(* IEC 61131-3 sources: vscode-st/examples, 13 files *)

(* ---- 02-function.st ---- *)
/* 02-function.st — FUNCTION with return type

   Demonstrates FUNCTION declaration with VAR_INPUT, local VAR, return value,
   RETURN statement (early exit), and function body with expressions. */

FUNCTION AddValues : INT
VAR_INPUT
    a : INT;
    b : INT;
END_VAR
VAR
    temp : INT;
END_VAR

// Compute sum and return
temp := a + b;

// Early RETURN guard — skips rest if condition met
IF temp > 1000 THEN
    AddValues := 0;
    RETURN;
END_IF;

AddValues := temp;

END_FUNCTION

(* ---- 03-function-block.st ---- *)
/* 03-function-block.st — FUNCTION_BLOCK

   Demonstrates FUNCTION_BLOCK with VAR_INPUT, VAR_OUTPUT, VAR,
   internal state logic, and ACTION definitions. */

FUNCTION_BLOCK CounterFB
VAR_INPUT
    enable  : BOOL;
    reset   : BOOL;
    maxVal  : INT := 100;
END_VAR
VAR_OUTPUT
    overflow : BOOL;
    current  : INT;
END_VAR
VAR
    internal : INT;
END_VAR

IF reset THEN
    internal := 0;
    current  := 0;
    overflow := FALSE;
ELSIF enable THEN
    IF internal < maxVal THEN
        internal := internal + 1;
    ELSE
        overflow := TRUE;
    END_IF;
    current := internal;
END_IF;

END_FUNCTION_BLOCK

FUNCTION_BLOCK MotorWithActions
VAR_INPUT
    startCmd : BOOL;
    stopCmd  : BOOL;
    speed    : REAL;
END_VAR
VAR_OUTPUT
    running    : BOOL;
    currentRPM : REAL;
END_VAR
VAR
    rampStep : REAL := 10.0;
END_VAR

IF startCmd THEN
    StartRamp();
ELSIF stopCmd THEN
    StopRamp();
END_IF;

ACTION StartRamp
    IF NOT running THEN
        running := TRUE;
        currentRPM := 0.0;
    END_IF;
    IF currentRPM < speed THEN
        currentRPM := currentRPM + rampStep;
    END_IF;
END_ACTION

ACTION StopRamp
    IF currentRPM > 0.0 THEN
        currentRPM := currentRPM - rampStep;
    ELSE
        running := FALSE;
        currentRPM := 0.0;
    END_IF;
END_ACTION

END_FUNCTION_BLOCK

(* ---- 04-namespace.st ---- *)
/* 04-namespace.st — NAMESPACE

   Demonstrates NAMESPACE containing multiple POU definitions.
   Namespaces group related POUs and provide name scoping. */

NAMESPACE MotorControl

    FUNCTION CalculateSpeed : REAL
    VAR_INPUT
        rpm     : INT;
        gearRatio : REAL;
    END_VAR
    VAR
        result : REAL;
    END_VAR
    result := INT_TO_REAL(rpm) * gearRatio;
    CalculateSpeed := result;
    END_FUNCTION

    PROGRAM MotorRunner
    VAR
        speed   : REAL;
        running : BOOL;
    END_VAR
    speed := CalculateSpeed(rpm := 1500, gearRatio := 3.14);
    IF running THEN
        speed := speed * 1.05;
    END_IF;
    END_PROGRAM

    FUNCTION_BLOCK PIDController
    VAR_INPUT
        setpoint : REAL;
        actual   : REAL;
        kp       : REAL := 1.0;
    END_VAR
    VAR_OUTPUT
        output : REAL;
    END_VAR
    VAR
        error : REAL;
    END_VAR
    error := setpoint - actual;
    output := kp * error;
    END_FUNCTION_BLOCK

END_NAMESPACE

(* ---- 06-class.st ---- *)
/* 06-class.st — CLASS, METHOD, PROPERTY (IEC 61131-3 OOP)

   Demonstrates CLASS declarations with access modifiers (PUBLIC, PRIVATE,
   PROTECTED, INTERNAL), ABSTRACT/FINAL/OVERRIDE method modifiers,
   PROPERTY with GET/SET, EXTENDS, and IMPLEMENTS. */

CLASS MotorBase IMPLEMENTS IMotor
    VAR
        _speed    : REAL;
        _enabled  : BOOL;
        _name     : STRING := 'MotorBase';
    END_VAR

    METHOD PUBLIC Start : BOOL
        _enabled := TRUE;
        Start := TRUE;
    END_METHOD

    METHOD PUBLIC Stop : BOOL
        _enabled := FALSE;
        _speed := 0.0;
        Stop := TRUE;
    END_METHOD

    METHOD PUBLIC SetSpeed : BOOL
    VAR_INPUT
        newSpeed : REAL;
    END_VAR
        IF _enabled THEN
            _speed := LIMIT(0.0, newSpeed, _maxSpeed);
            SetSpeed := TRUE;
        ELSE
            SetSpeed := FALSE;
        END_IF;
    END_METHOD

    METHOD PROTECTED GetMaxSpeed : REAL
        GetMaxSpeed := _maxSpeed;
    END_METHOD

END_CLASS

CLASS AdvancedMotor EXTENDS MotorBase IMPLEMENTS IAdvancedMotor
    VAR PRIVATE
        _accelRate : REAL := 5.0;
        _decelRate : REAL := 10.0;
        _targetSpeed : REAL;
    END_VAR

    VAR PUBLIC
        status : STRING := 'idle';
    END_VAR

    // Override the Start method
    METHOD PUBLIC OVERRIDE Start : BOOL
        status := 'ramping';
        Start := SUPER.Start();
    END_METHOD

    // Abstract method that must be implemented
    METHOD PUBLIC ABSTRACT Diagnose : STRING
    END_METHOD

    METHOD PUBLIC FINAL GetConfig : STRING
        GetConfig := CONCAT('Motor: ', _name);
    END_METHOD

    // Property with getter and setter
    PROPERTY PUBLIC TargetSpeed : REAL
        GET
            TargetSpeed := _targetSpeed;
        END_GET
        SET
            _targetSpeed := LIMIT(0.0, TargetSpeed, SUPER.GetMaxSpeed());
        END_SET
    END_PROPERTY

    // Read-only property (getter only)
    PROPERTY PUBLIC IsRunning : BOOL
        GET
            IsRunning := _enabled AND (_speed > 0.0);
        END_GET
    END_PROPERTY

    METHOD INTERNAL RampToTarget : BOOL
        IF _speed < _targetSpeed THEN
            _speed := _speed + _accelRate;
            IF _speed > _targetSpeed THEN
                _speed := _targetSpeed;
            END_IF;
        ELSIF _speed > _targetSpeed THEN
            _speed := _speed - _decelRate;
            IF _speed < _targetSpeed THEN
                _speed := _targetSpeed;
            END_IF;
        END_IF;
        status := CONCAT('speed: ', REAL_TO_STRING(_speed));
        RampToTarget := TRUE;
    END_METHOD

END_CLASS

(* ---- 07-interface.st ---- *)
/* 07-interface.st — INTERFACE with METHOD signatures

   Demonstrates INTERFACE declarations with METHOD signatures (no body)
   and IMPLEMENTS relationship with CLASS / FUNCTION_BLOCK. */

INTERFACE IMotor
    METHOD Start : BOOL
    END_METHOD

    METHOD Stop : BOOL
    END_METHOD

    METHOD SetSpeed : BOOL
    VAR_INPUT
        newSpeed : REAL;
    END_VAR
    END_METHOD

    METHOD GetName : STRING
    END_METHOD
END_INTERFACE

INTERFACE IAdvancedMotor EXTENDS IMotor
    METHOD Diagnose : STRING
    END_METHOD

    METHOD GetEfficiency : REAL
    VAR_INPUT
        loadPercent : INT;
    END_VAR
    END_METHOD

    METHOD EmergencyStop : BOOL
    END_METHOD
END_INTERFACE

INTERFACE ISerializable
    METHOD Serialize : STRING
    END_METHOD

    METHOD Deserialize : BOOL
    VAR_IN_OUT
        data : STRING;
    END_VAR
    END_METHOD
END_INTERFACE

// A function block implementing multiple interfaces
FUNCTION_BLOCK SmartMotor IMPLEMENTS IAdvancedMotor, ISerializable
    VAR
        _speed       : REAL;
        _enabled     : BOOL;
        _serialized  : STRING;
    END_VAR

    METHOD PUBLIC Start : BOOL
        _enabled := TRUE;
        Start := TRUE;
    END_METHOD

    METHOD PUBLIC Stop : BOOL
        _enabled := FALSE;
        _speed := 0.0;
        Stop := TRUE;
    END_METHOD

    METHOD PUBLIC SetSpeed : BOOL
    VAR_INPUT
        newSpeed : REAL;
    END_VAR
        _speed := newSpeed;
        SetSpeed := TRUE;
    END_METHOD

    METHOD PUBLIC GetName : STRING
        GetName := 'SmartMotor';
    END_METHOD

    METHOD PUBLIC Diagnose : STRING
        Diagnose := CONCAT('Speed=', REAL_TO_STRING(_speed));
    END_METHOD

    METHOD PUBLIC GetEfficiency : REAL
    VAR_INPUT
        loadPercent : INT;
    END_VAR
        GetEfficiency := 0.85;
    END_METHOD

    METHOD PUBLIC EmergencyStop : BOOL
        _enabled := FALSE;
        _speed := 0.0;
        EmergencyStop := TRUE;
    END_METHOD

    METHOD PUBLIC Serialize : STRING
        Serialize := CONCAT('SmartMotor:', REAL_TO_STRING(_speed));
    END_METHOD

    METHOD PUBLIC Deserialize : BOOL
    VAR_IN_OUT
        data : STRING;
    END_VAR
        Deserialize := TRUE;
    END_METHOD

END_FUNCTION_BLOCK

(* ---- 10-var-blocks.st ---- *)
/* 10-var-blocks.st — All VAR block variants

   Demonstrates every VAR keyword variant from the grammar: VAR, VAR_INPUT,
   VAR_OUTPUT, VAR_IN_OUT, VAR_GLOBAL with qualifiers (RETAIN, PERSISTENT,
   CONSTANT), AT addresses, comma-separated declarations, and VAR_EXTERNAL
   inside a POU. */

// Global variable block — available across the project
VAR_GLOBAL
    gSystemTick  : DINT;
    gMaxSpeed    : REAL    := 5000.0;
    gMachineName : STRING  := 'PLC001';
END_VAR

// Retained global — survives power cycle
VAR_GLOBAL RETAIN
    gRuntimeHours : DINT;
    gCycleCount   : DWORD;
END_VAR

// Persistent global — survives cold reset
VAR_GLOBAL PERSISTENT
    gSerialNumber : STRING  := 'SN-0001';
    gCalibration  : REAL    := 1.0;
END_VAR

// Constant global
VAR_GLOBAL CONSTANT
    gPI           : REAL    := 3.14159265359;
    gMaxMotors    : INT     := 8;
    gVersion      : STRING  := 'v2.0.0';
END_VAR

FUNCTION_BLOCK VarBlockDemo
    // Standard local variables
    VAR
        localCounter : INT;
        localFlag    : BOOL;
    END_VAR

    // Temporary — not retained across cycles
    VAR
        tempCalc     : REAL;
        tempString   : STRING;
    END_VAR

    // Input variables
    VAR_INPUT
        inEnable      : BOOL;
        inSpeedRef    : REAL;
    END_VAR

    // Output variables
    VAR_OUTPUT
        outActive     : BOOL;
        outSpeed      : REAL;
        outErrorCode  : WORD;
    END_VAR

    // In/Out (reference) variables
    VAR_IN_OUT
        ioPosition    : REAL;
        ioState       : DINT;
    END_VAR

    // AT address — direct I/O mapping
    VAR
        startButton   AT %IX0.0 : BOOL;
        stopButton    AT %IX0.1 : BOOL;
        eStopInput    AT %IX0.2 : BOOL;
        motorOutput   AT %QX1.0 : BOOL;
        analogInput   AT %IW2   : INT;
        analogOutput  AT %QW3   : INT;
    END_VAR

    // Multiple named variables comma-separated
    VAR
        x, y, z : REAL;
        i, j, k : INT    := 0;
        ok, err : BOOL;
    END_VAR

    // Initialized variables with various types
    VAR
        intVar     : INT    := 42;
        realVar    : REAL   := 3.14;
        boolVar    : BOOL   := TRUE;
        strVar     : STRING := 'initial';
        timeVar    : TIME   := T#1s500ms;
    END_VAR

    // External variable references — must be inside a POU
    VAR_EXTERNAL
        gSystemTick  : DINT;
        gMaxSpeed    : REAL;
        gCycleCount  : DWORD;
    END_VAR

    // Logic using the var blocks
    IF inEnable AND startButton AND NOT stopButton THEN
        outActive := TRUE;
        outSpeed := LIMIT(0.0, inSpeedRef, gMaxSpeed);
        motorOutput := TRUE;
        localCounter := localCounter + 1;
    ELSE
        outActive := FALSE;
        outSpeed := 0.0;
        motorOutput := FALSE;
    END_IF;

    ioPosition := ioPosition + (inSpeedRef * 0.01);

END_FUNCTION_BLOCK

(* ---- 14-try-catch.st ---- *)
/* 14-try-catch.st — Exception handling

   Demonstrates __TRY, __CATCH, __FINALLY, __ENDTRY blocks.
   These are vendor-specific extensions (primarily Beckhoff/Codesys)
   for structured exception handling. */

FUNCTION TryCatchDemo : INT
VAR_INPUT
    denominator : INT;
END_VAR
VAR
    result      : INT;
    errorFlag   : BOOL;
    errorMsg    : STRING;
END_VAR

__TRY
    // Guarded code block
    result := 100 / denominator;
    errorFlag := FALSE;
    errorMsg := '';
__CATCH
    // Exception handler — runs if __TRY block throws
    result := 0;
    errorFlag := TRUE;
    errorMsg := 'Division by zero or other error';
__FINALLY
    // Always runs — cleanup code
    // (e.g., close file handles, reset flags)
    TryCatchDemo := result;
__ENDTRY

END_FUNCTION

FUNCTION_BLOCK FileProcessor
VAR_INPUT
    fileName : STRING;
END_VAR
VAR_OUTPUT
    success  : BOOL;
    data     : DINT;
END_VAR
VAR
    fileHandle : DINT;
    buffer     : DINT;
END_VAR

success := FALSE;

__TRY
    fileHandle := SysFileOpen(fileName, 'r');
    __TRY
        // Nested try block for read operation
        buffer := SysFileRead(fileHandle);
        data := buffer;
    __CATCH
        data := 0;
    __FINALLY
        SysFileClose(fileHandle);
    __ENDTRY
    success := TRUE;
__CATCH
    success := FALSE;
    data := 0;
__FINALLY
    // Ensure file is closed even if outer try fails
    IF fileHandle <> 0 THEN
        SysFileClose(fileHandle);
    END_IF;
__ENDTRY

END_FUNCTION_BLOCK

(* ---- 01-program.st ---- *)
(* 01-program.st — Simple PROGRAM

   Demonstrates the most fundamental ST unit: a PROGRAM with VAR blocks,
   assignments, an IF statement, and function calls. Also shows ACTION
   definitions within a PROGRAM. *)

PROGRAM MainProgram
VAR
    counter : INT := 0;
    limit   : INT := 100;
    running : BOOL := TRUE;
    result  : REAL;
END_VAR

// Initialization and main loop logic
running := TRUE;
counter := counter + 1;

IF counter >= limit THEN
    running := FALSE;
    counter := 0;
END_IF;

result := SIN(INT_TO_REAL(counter));

// Call actions from the main body
IF counter MOD 3 = 0 THEN
    IncrementAction();
ELSIF counter MOD 3 = 1 THEN
    DecrementAction();
ELSE
    ResetAction();
END_IF;

ACTION IncrementAction
    counter := counter + 1;
    running  := TRUE;
END_ACTION

ACTION DecrementAction
    counter := counter - 1;
    IF counter < 0 THEN
        counter := 0;
    END_IF;
END_ACTION

ACTION ResetAction
    counter := 0;
    running  := FALSE;
END_ACTION

END_PROGRAM

(* ---- 05-types.st ---- *)
/* 05-types.st — TYPE declarations

   Demonstrates TYPE with STRUCT, ENUM, UNION, alias (ARRAY),
   and subrange-style type restrictions. */

// Alias — simple type renaming
TYPE SpeedType : REAL; END_TYPE

// Alias with default value
TYPE MaxLimit : INT := 100; END_TYPE

// Alias referencing another type
TYPE MotorSpeed : SpeedType; END_TYPE

// Enumeration
TYPE MotorState : (Idle, Running, Stopped, Error) := Idle; END_TYPE

// Enumeration with explicit values
TYPE ErrorCode : (
    NoError     := 0,
    Timeout     := 100,
    Overcurrent := 200,
    ThermalTrip := 300
) := NoError; END_TYPE

// Structure
TYPE MotorConfig : STRUCT
    maxRPM       : INT     := 3000;
    accelRate    : REAL    := 1.5;
    enabled      : BOOL    := TRUE;
    state        : MotorState;
    faultCode    : ErrorCode;
    name         : STRING  := 'Motor1';
END_STRUCT; END_TYPE

// Union
TYPE SensorValue : UNION
    asInteger : DINT;
    asReal    : REAL;
    asWord    : WORD;
END_UNION; END_TYPE

// Array type alias
TYPE AnalogArray : ARRAY[0..7] OF INT; END_TYPE

// Multi-dimensional array alias
TYPE Matrix3x3 : ARRAY[0..2, 0..2] OF REAL; END_TYPE

PROGRAM TypeUser
VAR
    speed    : MotorSpeed := 3.14;
    cfg      : MotorConfig;
    state    : MotorState := MotorState.Running;
    readings : AnalogArray;
    matrix   : Matrix3x3;
    sensor   : SensorValue;
END_VAR
speed := cfg.accelRate;
END_PROGRAM

(* ---- 08-expressions.st ---- *)
/* 08-expressions.st — All operators, function calls, IEC addresses

   Demonstrates the full expression syntax of IEC 61131-3 ST.
   Arithmetic: + - * / MOD, comparison: = <> < > <= >=,
   logical: AND OR XOR NOT, function calls, parenthesized expressions,
   IEC hardware addresses (%IX0.0, %QW5, etc.), and type conversions. */

PROGRAM ExpressionDemo
VAR
    a, b, c   : INT    := 0;
    x, y, z   : REAL   := 0.0;
    flag1     : BOOL;
    flag2     : BOOL   := TRUE;
    inputBit  : BOOL;
    outputBit AT %QX0.0 : BOOL;
    sensor    AT %IW2  : WORD;
    result    : DINT;
END_VAR

// --- Arithmetic operators ---
a := 10 + 5;                    // Addition
b := 20 - 3;                    // Subtraction
c := a * b;                     // Multiplication
x := REAL#100.0 / REAL#3.0;     // Division
y := REAL_TO_INT(a) MOD 3;      // Modulo

// --- Comparison operators ---
flag1 := a = b;                 // Equal
flag1 := a <> b;                // Not equal
flag1 := a < b;                 // Less than
flag1 := a > b;                 // Greater than
flag1 := a <= b;                // Less than or equal
flag1 := a >= b;                // Greater than or equal

// --- Logical operators ---
flag1 := flag2 AND (a > 5);
flag1 := flag1 OR flag2;
flag1 := flag1 XOR flag2;
flag1 := NOT flag1;

// --- Parenthesized compound expressions ---
result := (a + b) * (c - 1) / 2;
flag1  := (a > 0) AND ((b < 10) OR (c = 5));

// --- Function calls ---
y := SIN(x);
y := COS(REAL#0.5);
y := SQRT(REAL#25.0);
z := ABS(REAL#-42.0);
result := MAX(a, b);
result := MIN(INT_TO_DINT(a), INT_TO_DINT(b));
result := LIMIT(MN := 0, IN := c, MX := 100);
result := SEL(G := flag2, IN0 := a, IN1 := b);

// --- Named and positional parameters ---
z := LIMIT(0, x, 100);                        // Positional
z := LIMIT(MN := 0.0, IN := x, MX := 100.0);  // Named assignment (:=)
z := LIMIT(MN := 0.0, IN => x, MX => 100.0);  // Named mapping (=>), Beckhoff-style

// --- Type conversion functions ---
// Format: sourceType_TO_targetType(value)
a := REAL_TO_INT(z);
x := INT_TO_REAL(a);
b := WORD_TO_INT(sensor);
result := DINT_TO_INT(result);

// --- NaN/Infinity sentinel values ---
c := INT#5;
x := REAL#3.14;

// --- Parenthesized sub-expressions with operators ---
x := (a + b) * (y - z);
flag1 := (a > b) AND ((c < 10) XOR (flag2));

// --- Multi-assignment (chained) ---
a := b := c := 0;

// --- IEC address expressions ---
// Direct I/O addressing — IEC 61131-3 hardware addresses
inputBit := %IX0.0;        // Input bit channel 0, bit 0
inputBit := %IX1.7;        // Input bit channel 1, bit 7
outputBit := flag1;         // Write to output via AT var

// Extended addressing — memory markers, multi-level dotted
%MW10 := 100;               // Memory word 10
%MD20 := 200;               // Memory double-word 20
%ML100 := 300;              // Memory long-word 100
%QX0.0 := TRUE;             // Output bit
%QW5 := WORD#16#00FF;       // Output word
%QD3 := DWORD#0;            // Output double-word
%QL7 := LWORD#0;            // Output long-word
%ID0.1.2 := 42;             // Input double-word, nested subaddress

// Reading analog input word via AT variable
result := sensor AND WORD#16#00FF;

// Assignment via IEC address AT variable
flag2 := %IX0.0;

// --- Chained comparisons / expressions ---
IF (a > 0) AND (b < 100) THEN
    c := c + 1;
END_IF;

// --- RETURN statement (inside FUNCTION context) ---
// Used in 03-function-block.st and 15-multi-file/motor_fb.st

END_PROGRAM

(* ---- 09-control-flow.st ---- *)
/* 09-control-flow.st — All control flow constructs

   Demonstrates IF/ELSIF/ELSE, CASE, FOR (with BY), WHILE, REPEAT,
   EXIT, CONTINUE, and RETURN. */

PROGRAM ControlFlowDemo
VAR
    i, j          : INT    := 0;
    value         : INT    := 42;
    flag          : BOOL   := FALSE;
    sumFor        : INT    := 0;
    sumWhile      : INT    := 0;
    sumRepeat     : INT    := 0;
    state         : INT    := 0;
    result        : STRING;
END_VAR

// --- IF / ELSIF / ELSE ---
IF value < 0 THEN
    result := 'negative';
ELSIF value = 0 THEN
    result := 'zero';
ELSIF value < 100 THEN
    result := 'small positive';
ELSE
    result := 'large positive';
END_IF;

// --- Nested IF ---
IF flag THEN
    IF value > 50 THEN
        result := 'flag and high';
    END_IF;
END_IF;

// --- CASE ---
CASE state OF
    0:
        result := 'idle';
    1:
        result := 'running';
    2:
        result := 'paused';
    3:
        result := 'error';
    ELSE
        result := 'unknown state';
END_CASE;

// --- CASE with ranges (integer values) ---
CASE value OF
    0..9:
        result := '0-9';
    10..19:
        result := '10-19';
    20, 30, 40:
        result := '20 or 30 or 40';
    ELSE
        result := 'other';
END_CASE;

// --- FOR loop ---
// Basic FOR with TO
sumFor := 0;
FOR i := 1 TO 10 DO
    sumFor := sumFor + i;
END_FOR;

// FOR with BY (step)
sumFor := 0;
FOR i := 0 TO 100 BY 5 DO
    sumFor := sumFor + i;
END_FOR;

// Nested FOR loops
sumFor := 0;
FOR i := 1 TO 3 DO
    FOR j := 1 TO 3 DO
        sumFor := sumFor + (i * j);
    END_FOR;
END_FOR;

// FOR with EXIT
sumFor := 0;
FOR i := 1 TO 100 DO
    sumFor := sumFor + i;
    IF sumFor > 1000 THEN
        EXIT;
    END_IF;
END_FOR;

// --- WHILE loop ---
sumWhile := 0;
i := 0;
WHILE i < 10 DO
    i := i + 1;
    sumWhile := sumWhile + i;
END_WHILE;

// WHILE with CONTINUE (skip even numbers)
sumWhile := 0;
i := 0;
WHILE i < 20 DO
    i := i + 1;
    IF i MOD 2 = 0 THEN
        CONTINUE;
    END_IF;
    sumWhile := sumWhile + i;
END_WHILE;

// WHILE with EXIT (early termination)
i := 0;
WHILE TRUE DO
    i := i + 1;
    IF i >= 5 THEN
        EXIT;
    END_IF;
END_WHILE;

// --- REPEAT loop ---
sumRepeat := 0;
i := 0;
REPEAT
    i := i + 1;
    sumRepeat := sumRepeat + i;
UNTIL i >= 10
END_REPEAT;

// REPEAT with EXIT
i := 0;
REPEAT
    i := i + 1;
    IF i > 50 THEN
        EXIT;
    END_IF;
UNTIL FALSE
END_REPEAT;

// --- Standalone EXIT as loop-break body ---
i := 0;
WHILE TRUE DO
    EXIT;
END_WHILE;

// Standalone CONTINUE as loop-break body
i := 0;
FOR i := 1 TO 1 DO
    CONTINUE;
END_FOR;

// --- RETURN (inside FUNCTION context) ---
// In a FUNCTION, RETURN exits with the function's current return value.

END_PROGRAM

(* ---- 12-strings-comments.st ---- *)
// 12-strings-comments.st — String literals and comment forms
// Demonstrates single-quoted strings, double-quoted strings,
// escape sequences, // line comments, (* *) block comments,
// /* */ block comments, nested comments, and comments in expressions.

// This is a single-line comment
// All comment types in one file

PROGRAM StringCommentDemo
VAR
    name        : STRING := 'Hello World';              // Single-quoted string
    message     : STRING := "Hello World";              // Double-quoted string
    emptyStr    : STRING := '';                         // Empty single-quoted
    emptyDbl    : STRING := "";                         // Empty double-quoted
    special     : STRING := 'It''s working';            // Escaped single quote
    dblEscape   : STRING := "He said ""yes""";          // Escaped double quote
    dollars     : STRING := 'Cost: $100.00';            // Dollar sign in string
    path        : WSTRING := "C:\Path\To\File";         // Double-quoted WSTRING
    dollarPath  : STRING := '$$C:\Path$$';                // Dollar signs in string
    concatStr   : STRING;
    numeric     : INT    := 42;
END_VAR

(* This is a block comment using (* *) delimiters
   It can span multiple lines.
*)

/* This is a block comment using /* */ delimiters
   Also can span multiple lines.
*/

(* Nested block comment: (* inner comment *) back to outer *)
(* Another nested: (* level 1: (* level 2: deep *) back *) done *)

// --- Comments in expressions ---
name := 'Hello' (* middle comment *) CONCAT ' World';   // Commented concat
name := CONCAT('Part1', (* between params *) 'Part2');

// --- Comments on code lines ---
numeric := 0; // trailing line comment
numeric :=
    (* block comment between token and value *)
    42;

// --- Strings with special content ---
name    := 'Special chars: @#$%^&*()_+-=[]{}|;:,.<>?/';
message := "Numbers: 1234567890";
name    := 'Mixed with ''quotes'' inside';
message := "Mixed with ""quotes"" inside";

// --- Concatenation ---
concatStr := CONCAT('Hello, ', 'World!');
concatStr := CONCAT(CONCAT('Nested ', 'concat '), 'call');

// --- WSTRING (wide string) ---
// path := WSTRING#"Unicode";
// path := WSTRING#'Wide';

// --- Comment-only areas (should not affect parsing) ---
(*
    Entire block of comments
    No code here at all
    Just documentation
*)
/*
    Another comment-only block
    With /* nested */ inside
*/

END_PROGRAM

(* ---- 13-data-types.st ---- *)
/* 13-data-types.st — All standard data types

   Demonstrates every IEC 61131-3 elementary data type:
   integers, reals, strings, time/dates, bit/byte/word types.
   Also: arrays, initial values, subrange types. */

PROGRAM DataTypeDemo
VAR
    // --- Boolean and bit strings ---
    b1, b2     : BOOL   := TRUE;
    byteVal    : BYTE   := BYTE#16#FF;
    wordVal    : WORD   := WORD#16#ABCD;
    dwordVal   : DWORD  := DWORD#16#DEADBEEF;
    lwordVal   : LWORD  := LWORD#16#0123456789ABCDEF;

    // --- Signed integers ---
    sVal       : SINT   := SINT#-128;          // 8-bit signed
    iVal       : INT    := -32768;             // 16-bit signed
    dVal       : DINT   := -2147483648;        // 32-bit signed
    lVal       : LINT   := -9223372036854775808; // 64-bit signed

    // --- Unsigned integers ---
    usVal      : USINT  := 255;                // 8-bit unsigned
    uiVal      : UINT   := 65535;              // 16-bit unsigned
    udVal      : UDINT  := 4294967295;         // 32-bit unsigned
    ulVal      : ULINT  := 18446744073709551615; // 64-bit unsigned

    // --- Floating point ---
    rVal       : REAL   := REAL#3.14159265;     // 32-bit float
    lrVal      : LREAL  := LREAL#2.718281828459045; // 64-bit float

    // --- Strings ---
    strVal     : STRING := 'IEC 61131-3';       // Variable-length string
    str80      : STRING(80) := 'Fixed 80';      // Fixed-length string (80 chars)
    wstrVal    : WSTRING := "Wide string";      // Unicode wide string
    wstrFixed  : WSTRING(255) := "Fixed wide";  // Fixed-length wide string

    // --- Time and date types ---
    timeVal    : TIME    := T#5s;               // Duration
    timeMs     : TIME    := T#500ms;             // Milliseconds
    timeUs     : TIME    := T#100us;             // Microseconds
    timeNs     : TIME    := T#50ns;              // Nanoseconds
    timeH      : TIME    := T#1h30m;            // Hours and minutes
    timeD      : TIME    := T#2d6h;             // Days and hours
    timeComplex: TIME    := T#1d2h30m15s500ms;  // Combined

    todVal     : TOD     := TOD#12:30:45.500;   // Time of day
    todShort   : TOD     := TOD#08:00:00;        // Time of day simple
    dateVal    : DATE    := DATE#2024-01-15;     // Date
    dtVal      : DT      := DT#2024-01-15-12:30:45; // Date and time
    ltodVal    : LTOD    := LTOD#12:30:45.123456789; // Long TOD
    ldateVal   : LDATE   := LDATE#2024-01-15;   // Long date
    ldtVal     : LDT     := LDT#2024-01-15-12:30:45.123456789; // Long DT

    // --- ANY type (generic) --- Not typically used in declarations

    // --- Subrange types ---
    smallUInt  : UINT (0..100);                     // Subrange: 0 to 100
    percent    : INT (0..100) := 50;                 // Subrange with init
    tinyInt    : SINT (-10..10);                     // Negative subrange

    // --- Arrays ---
    arr1D      : ARRAY[0..9] OF INT;                  // 1D array of INT
    arr2D      : ARRAY[0..3, 0..3] OF REAL;           // 2D array
    arr3D      : ARRAY[0..1, 0..1, 0..1] OF BOOL;     // 3D array
    arrStr     : ARRAY[1..5] OF STRING(20);            // 1D array of strings
    arrInit    : ARRAY[0..2] OF INT := [10, 20, 30];  // Array with initializer
    arrInit2D  : ARRAY[0..1, 0..1] OF INT := [1, 2, 3, 4]; // 2D initializer

    // --- Structured types (see 05-types.st for TYPE-based) ---

    // --- Aliased types (any DT variant can be used as type) ---
    intResult  : DINT;
    realResult : LREAL;
    wordResult : WORD;
END_VAR

// --- Operations on various types ---
intResult := iVal + dVal;                    // Mixed integer ops
realResult := REAL_TO_LREAL(rVal) * lrVal;   // Mixed real ops
wordResult := wordVal OR WORD#16#00FF;       // Bitwise on word

timeVal := timeVal + T#1s;                  // Time arithmetic
timeVal := timeComplex - T#500ms;            // Time subtraction

arr1D[0] := 42;                              // Array access
arr2D[1, 2] := 3.14;                         // Multi-dim array access

END_PROGRAM
